// Mitsubishi GX Works2 project: ProMayMai   PLC: FX1S

PROGRAM MAIN
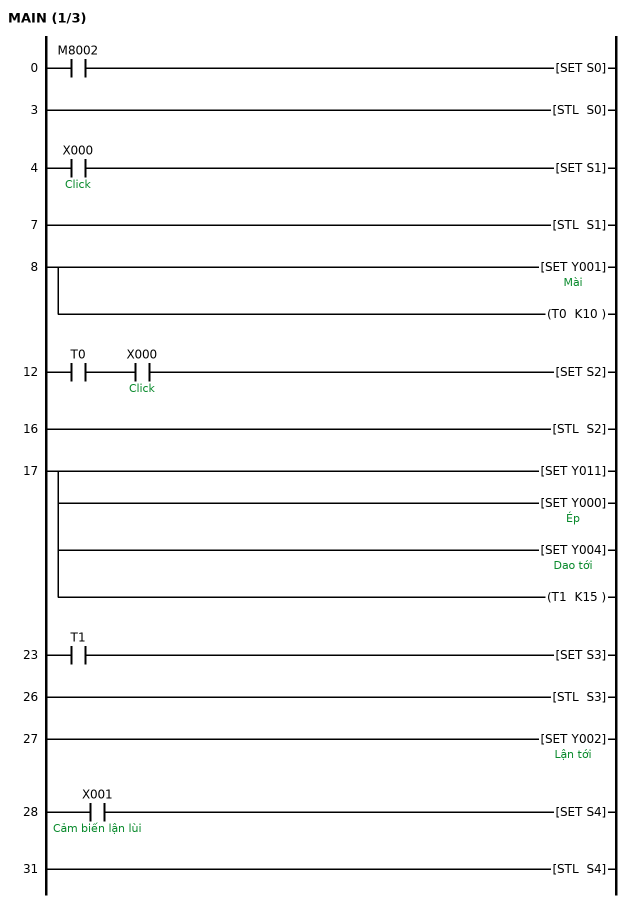
0     LD      M8002
      SET     S0
3     STL     S0
4     LD      X000  ; Click
      SET     S1
7     STL     S1
8     SET     Y001  ; Mài
      OUT     T0 K10
12    LD      T0
      AND     X000  ; Click
      SET     S2
16    STL     S2
17    SET     Y011
      SET     Y000  ; Ép
      SET     Y004  ; Dao tới
      OUT     T1 K15
23    LD      T1
      SET     S3
26    STL     S3
27    SET     Y002  ; Lận tới
28    LD      X001  ; Cảm biến lận lùi
      SET     S4
31    STL     S4
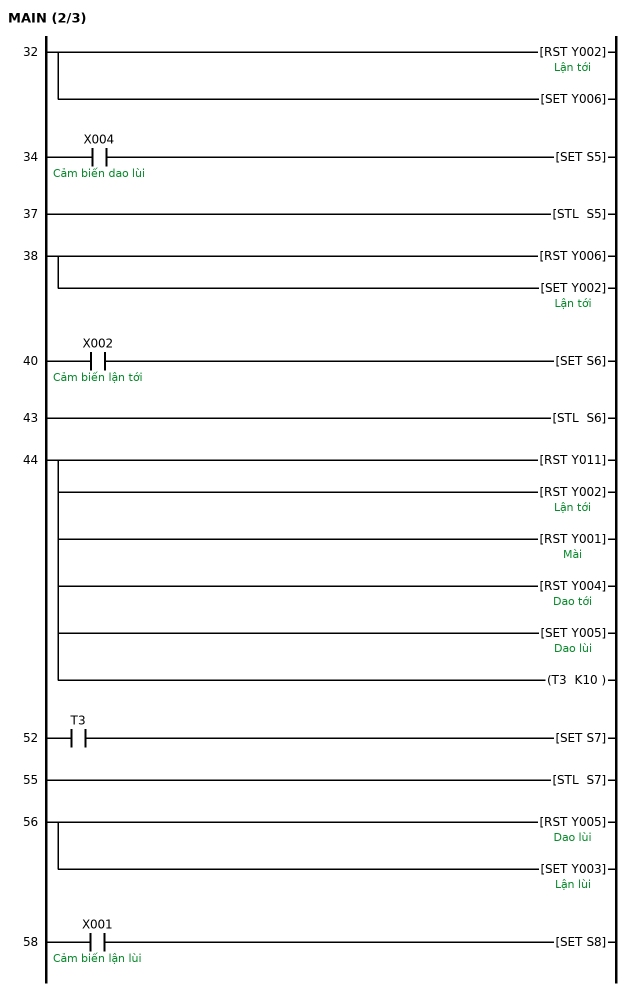
32    RST     Y002  ; Lận tới
      SET     Y006
34    LD      X004  ; Cảm biến dao lùi
      SET     S5
37    STL     S5
38    RST     Y006
      SET     Y002  ; Lận tới
40    LD      X002  ; Cảm biến lận tới
      SET     S6
43    STL     S6
44    RST     Y011
      RST     Y002  ; Lận tới
      RST     Y001  ; Mài
      RST     Y004  ; Dao tới
      SET     Y005  ; Dao lùi
      OUT     T3 K10
52    LD      T3
      SET     S7
55    STL     S7
56    RST     Y005  ; Dao lùi
      SET     Y003  ; Lận lùi
58    LD      X001  ; Cảm biến lận lùi
      SET     S8
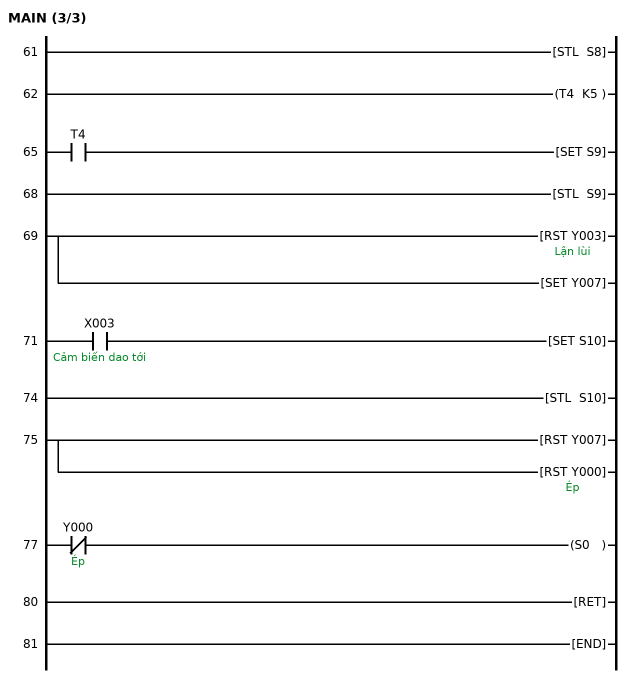
61    STL     S8
62    OUT     T4 K5
65    LD      T4
      SET     S9
68    STL     S9
69    RST     Y003  ; Lận lùi
      SET     Y007
71    LD      X003  ; Cảm biến dao tới
      SET     S10
74    STL     S10
75    RST     Y007
      RST     Y000  ; Ép
77    LDI     Y000  ; Ép
      OUT     S0
80    RET
81    END
END_PROGRAM
